DATA_BLOCK "M1_instance_DB"
{ DB_Accessible_From_OPC_UA := 'FALSE' ;
 S7_Optimized_Access := 'TRUE' }
AUTHOR : Frj
VERSION : 0.1
NON_RETAIN
"device_control"

BEGIN
   M_out.set_mode_op := 16#03;

END_DATA_BLOCK

